// TIA Portal project "260605_V003_Wendeschütz_NotAus" (V17)

(* hardware
DEVICE "S7-1500/ET200MP-Station_1"  S7-1500 station
   slot 0: "Profilschiene_0"  Rack  6ES7 590-1***0-0AA0
   slot 0: "PM 70W 120/230VAC"  PM 70W 120/230VAC  6EP1332-4BA00
   slot 1: "PLC_1"  CPU 1516-3 PN/DP  6ES7 516-3AN02-0AB0  V2.9
      slot 3: "CPU-Display_1"  6ES7591-1BA00-0AA0
      slot 32768: "PROFINET-Schnittstelle_1"  X1
         slot 32769: "Port_1"  X1 P1
         slot 32770: "Port_2"  X1 P2
      slot 33024: "PROFINET-Schnittstelle_2"  X2
         slot 33025: "Port_1"  X2 P1
      slot 33280: "DP-Schnittstelle_1"  X3
      slot 34817: "Virtual CP interface port_1"  Virtual CP interface port  Virtual CP interface port
   slot 2: "DI 32x24VDC HF_1"  DI 32x24VDC HF  6ES7 521-1BL00-0AB0  V2.1
   slot 3: "DQ 32x24VDC/0.5A ST_1"  DQ 32x24VDC/0.5A ST  6ES7 522-1BL00-0AB0  V2.0
   slot 4: "AI 8xU/I/RTD/TC ST_1"  AI 8xU/I/RTD/TC ST  6ES7 531-7KF00-0AB0  V2.2
   slot 5: "AQ 4xU/I ST_1"  AQ 4xU/I ST  6ES7 532-5HD00-0AB0  V2.1
*)

// ===== PLC "PLC_1"  CPU 1516-3 PN/DP =====

VAR_GLOBAL   // PLC tag table "Standard-Variablentabelle"
   "S1Motor1_Aus" AT %E0.0 : Bool;
   "S2Motor1_Rechtslauf" AT %E0.1 : Bool;
   "S3Motor1_Linkslauf" AT %E0.2 : Bool;
   "Q1RL_Motor1Rechts" AT %A0.0 : Bool;   // Ansteuerung Schütz Motor 1 Rechtslauf
   "Q2LL_Motor1Linkslauf" AT %A0.1 : Bool;   // Ansteuerung Schütz Motor 1 Linkslauf
   "F1MSS_Motor1_NC" AT %E0.3 : Bool;
   "SpeicherM1RL" AT %M10.0 : Bool;
   "SpeicherM1LL" AT %M10.1 : Bool;
   "S5_NotAus_NC" AT %E0.5 : Bool;
   "S6_Reset_NA" AT %E0.6 : Bool;
   "NotAusOK" AT %M5.0 : Bool;
   "AlwaysFalse" AT %M0.0 : Bool;
END_VAR

FUNCTION "fc005_NotAus" : Void   // FC5, FBD
{ S7_Optimized_Access := 'TRUE' }
VERSION : 0.1
BEGIN

REGION Network 1
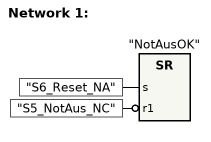
   IF "S6_Reset_NA" THEN
       "NotAusOK" := TRUE;   // SR flip-flop
   END_IF;
   IF NOT "S5_NotAus_NC" THEN "NotAusOK" := FALSE; END_IF;
END_REGION
END_FUNCTION

FUNCTION "fc050_AnsteuerungM1" : Void   // FC50, FBD
{ S7_Optimized_Access := 'TRUE' }
VERSION : 0.1
BEGIN

REGION Network 1: Ansteuerung Schütz Motor 1 Rechtslauf
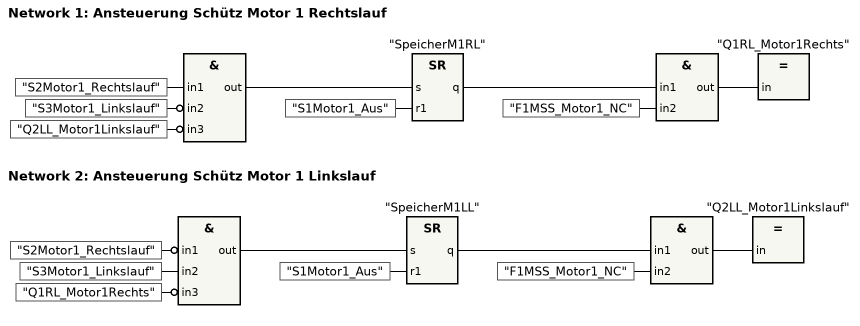
   IF "S2Motor1_Rechtslauf" AND NOT "S3Motor1_Linkslauf" AND NOT "Q2LL_Motor1Linkslauf" THEN
       "SpeicherM1RL" := TRUE;   // SR flip-flop
   END_IF;
   IF "S1Motor1_Aus" THEN "SpeicherM1RL" := FALSE; END_IF;
   "Q1RL_Motor1Rechts" := "SpeicherM1RL" AND "F1MSS_Motor1_NC";
END_REGION

REGION Network 2: Ansteuerung Schütz Motor 1 Linkslauf
   IF NOT "S2Motor1_Rechtslauf" AND "S3Motor1_Linkslauf" AND NOT "Q1RL_Motor1Rechts" THEN
       "SpeicherM1LL" := TRUE;   // SR flip-flop
   END_IF;
   IF "S1Motor1_Aus" THEN "SpeicherM1LL" := FALSE; END_IF;
   "Q2LL_Motor1Linkslauf" := "SpeicherM1LL" AND "F1MSS_Motor1_NC";
END_REGION
END_FUNCTION

ORGANIZATION_BLOCK "Main"   // OB1, FBD, ProgramCycle
TITLE = "Main Program Sweep (Cycle)"
{ S7_Optimized_Access := 'TRUE' }
VERSION : 0.1
   VAR_INPUT
      Initial_Call : Bool;   // Initial call of this OB
      Remanence : Bool;   // =True, if remanent data are available
   END_VAR
BEGIN

REGION Network 1
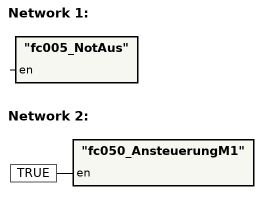
   "fc005_NotAus"();
END_REGION

REGION Network 2
   IF TRUE THEN "fc050_AnsteuerungM1"(); END_IF;
END_REGION
END_ORGANIZATION_BLOCK